{attribute 'GeneratedUsingTerminal: EJ9576-0000-0018'}
{attribute addProperty BoxType "EJ9576-0000-0018"}
{attribute addProperty Id "BCT_InputsAT %I*BCT_Inputs_8E55234D16WcStateAT %I*WcState_9091E0EB2InfoDataAT %I*InfoData_94A18F5E2"}
{attribute addProperty CRC "78208026"}
{attribute addProperty Size "20"}
TYPE EJ9576_04A95C1A EXTENDS EtcSlaveTerminalBase_947E5A46 :
STRUCT
	{attribute addProperty Name "BCT_Inputs"}
	BCT_Inputs : BCT_Inputs_8E55234D;
	{attribute addProperty Name "WcState"}
	WcState : WcState_9091E0EB;
	{attribute addProperty Name "InfoData"}
	InfoData : InfoData_94A18F5E;
END_STRUCT
END_TYPE

(* stored: Version 1.2.0.0, ProductVersion 3.1.4024.9
   DUT EJ9576_04A95C1A: Id {0cd1eaa4-359a-42a1-ab6d-d75ba7963671} *)
